PROGRAM SP_change
  VAR_OUTPUT
    wPrsHourSP_1 : WORD := 6;  (* Часы инициализации дневной уставки *)
    wPrsMinSP_1 : WORD;  (* Минуты инициализации дневной уставки *)
    wPrsHourSP_2 : WORD := 21;  (* Часы инициализации ночной уставки *)
    wPrsMinSP_2 : WORD;  (* Минуты инициализации ночной уставки *)
    wPrsHourSP_3 : WORD := 6;  (* Часы инициализации дневной зимней уставки *)
    wPrsMinSP_3 : WORD;  (* Минуты инициализации дневной зимней уставки *)
    wPrsHourSP_4 : WORD := 20;  (* Часы инициализации ночной зимней уставки *)
    wPrsMinSP_4 : WORD;  (* Минуты инициализации ночной зимней уставки *)
  END_VAR
  VAR_IN_OUT
    wPrsDayS : WORD;  (* День переключения на летний режим *)
    wPrsMonthS : WORD;  (* Месяц переключения на летний режим *)
    wPrsDayW : WORD;  (* День переключения на зимний режим *)
    wPrsMonthW : WORD;  (* Месяц переключения на зимний режим *)
  END_VAR
  VAR
    SP_in : REAL;  (* Входная уставка из контроллера *)
    SP_in2 : REAL;
    SP_old_man : REAL;
    write_sp : INT;
  END_VAR
  VAR_OUTPUT
    Summer : BOOL;
  END_VAR
  VAR_IN_OUT
    wCmdSP : WORD;  (* Слово на запись уставок *)
  END_VAR
  VAR_OUTPUT
    rPrsSP_1 : REAL;  (* Уставка давления №1 (летняя, дневная) *)
    rPrsSP_2 : REAL;  (* Уставка давления №2 (летняя, ночная) *)
    rPrsSP_3 : REAL;  (* Уставка давления №3 (зимняя, дневная) *)
    rPrsSP_4 : REAL;  (* Уставка давления №4 (зимняя, ночная) *)
    SP_target : REAL;
    SP : REAL;  (* Текущая уставка *)
  END_VAR
  VAR
    xPrsSP_N : BOOL;  (* Запись уставки по номеру *)
    xPrsSchedSP : BOOL;  (* Запись уставки по расписанию *)
    rem_auto_man : WORD := 3;  (* режим работы регулятора *)
    speed_limit : Speed_Lim;
    InputNum : Stat_to_num;
  END_VAR
  VAR_INPUT
    wNumSP : WORD;  (* Номер уставки *)
    rPrsDN : REAL;  (* Уставка давления день/ночь *)
    rPrsSched : REAL;  (* Уставка давления по расписанию *)
    rSP_manual : REAL;  (* Ручная уставка *)
    wPrsHourSP_N : WORD;  (* Часы инициализации уставки *)
    wPrsMinSP_N : WORD;  (* Минуты инициализации уставки *)
    xSCADA_Comm : BOOL;  (* Наличие связи со SCADA *)
    r_dSP : REAL;  (* скорость изменения уставки *)
  END_VAR

            wPrsMonthS:=LIMIT(1,wPrsMonthS,12);
wPrsMonthW:=LIMIT(1,wPrsMonthW,12);
wPrsDayS:=LIMIT(1, WORD_TO_UINT(wPrsDayS), QDay(y:=wYear , m:=WORD_TO_UINT(wPrsMonthS)));
wPrsDayW:=LIMIT(1, WORD_TO_UINT(wPrsDayW), QDay(y:=wYear , m:=WORD_TO_UINT(wPrsMonthW)));

IF wPrsMonthW > wPrsMonthS OR wPrsMonthW = wPrsMonthS AND wPrsDayW > wPrsDayS THEN
	IF wMonth>wPrsMonthW OR wMonth=wPrsMonthW AND wDay>=wPrsDayW OR wMonth<wPrsMonthS OR wMonth=wPrsMonthS AND wDay<wPrsDayS THEN
		Summer:=0;
		wCmdSP.10:=0;
	ELSIF wMonth>wPrsMonthS OR wMonth=wPrsMonthS AND wDay>=wPrsDayS THEN
		Summer:=1;
		wCmdSP.10:=1;
	END_IF
(*ELSE 
	END_IF*)
END_IF

///////////////////////////////Переключение уставок день/ночь/ Лето//////////////////////////
IF Summer THEN
IF wPrsHourSP_2>wPrsHourSP_1 OR wPrsHourSP_2=wPrsHourSP_1 AND wPrsMinSP_2>wPrsMinSP_1 THEN
	IF wHour>wPrsHourSP_2 OR wHour=wPrsHourSP_2 AND wMinute>=wPrsMinSP_2 OR wHour<wPrsHourSP_1 OR wHour=wPrsHourSP_1 AND wMinute<wPrsMinSP_1 THEN
		IF NOT write_sp.1 THEN
			write_sp:=0;
			SP_in:=rPrsSP_2;
			write_sp.1:=1;
		END_IF
	ELSIF wHour>wPrsHourSP_1 OR wHour=wPrsHourSP_1 AND wMinute>=wPrsMinSP_1 THEN
		IF NOT write_sp.0 THEN
			write_sp:=0;
			SP_in:=rPrsSP_1;
			write_sp.0:=1;
		END_IF
	END_IF
ELSE 
	IF wHour>wPrsHourSP_1 OR wHour=wPrsHourSP_1 AND wMinute>=wPrsMinSP_1 OR wHour<wPrsHourSP_2 OR wHour=wPrsHourSP_2 AND wMinute<wPrsMinSP_2 THEN
			IF NOT write_sp.2 THEN
			write_sp:=0;
			SP_in:=rPrsSP_1;
			write_sp.2:=1;
		END_IF
	ELSIF wHour>wPrsHourSP_2 OR wHour=wPrsHourSP_2 AND wMinute>=wPrsMinSP_2 THEN
		IF NOT write_sp.3 THEN
			write_sp:=0;
			SP_in:=rPrsSP_2;
			write_sp.3:=1;
		END_IF
	END_IF
END_IF
///////////////////////////////////////////////////////////////////////////////////////////////////
ELSE
///////////////////////////////Переключение уставок день/ночь/ Зима//////////////////////////
IF wPrsHourSP_4>wPrsHourSP_3 OR wPrsHourSP_4=wPrsHourSP_3 AND wPrsMinSP_4>wPrsMinSP_3 THEN
	IF wHour>wPrsHourSP_4 OR wHour=wPrsHourSP_4 AND wMinute>=wPrsMinSP_4 OR wHour<wPrsHourSP_3 OR wHour=wPrsHourSP_3 AND wMinute<wPrsMinSP_3 THEN
		IF NOT write_sp.5 THEN
			write_sp:=0;
			SP_in:=rPrsSP_4;
			write_sp.5:=1;
		END_IF
	ELSIF wHour>wPrsHourSP_3 OR wHour=wPrsHourSP_3 AND wMinute>=wPrsMinSP_3 THEN	
		IF NOT write_sp.4 THEN
			write_sp:=0;
			SP_in:=rPrsSP_3;
			write_sp.4:=1;
		END_IF
	END_IF
ELSE 
	IF wHour>wPrsHourSP_3 OR wHour=wPrsHourSP_3 AND wMinute>=wPrsMinSP_3 OR wHour<wPrsHourSP_4 OR wHour=wPrsHourSP_4 AND wMinute<wPrsMinSP_4 THEN
		IF NOT write_sp.6 THEN
			write_sp:=0;
			SP_in:=rPrsSP_3;
			write_sp.6:=1;
		END_IF
	ELSIF wHour>wPrsHourSP_4 OR wHour=wPrsHourSP_4 AND wMinute>=wPrsMinSP_4 THEN
		IF NOT write_sp.7 THEN
			write_sp:=0;
			SP_in:=rPrsSP_4;
			write_sp.7:=1;
		END_IF
	END_IF
END_IF
///////////////////////////////////////////////////////////////////////////////////////////////////
END_IF;

InputNum(in1:=wCmdSP.3,in2:=wCmdSP.4,in3:=wCmdSP.5);
rem_auto_man:=InputNum.out;

///////////////////////////////Ввод уставок из SCADA///////////////////////////
xPrsSP_N:=wCmdSP.0;
	IF xPrsSP_N THEN
		CASE wNumSP OF
			1: rPrsSP_1:=rPrsDN;
			wPrsHourSP_1:=wPrsHourSP_N;
			wPrsMinSP_1:=wPrsMinSP_N;
			2: rPrsSP_2:=rPrsDN;
			wPrsHourSP_2:=wPrsHourSP_N;
			wPrsMinSP_2:=wPrsMinSP_N;						
			3: rPrsSP_3:=rPrsDN;
			wPrsHourSP_3:=wPrsHourSP_N;
			wPrsMinSP_3:=wPrsMinSP_N;			
			4: rPrsSP_4:=rPrsDN;
			wPrsHourSP_4:=wPrsHourSP_N;
			wPrsMinSP_4:=wPrsMinSP_N;
		END_CASE
		xPrsSP_N:=0;
		wCmdSP.0:=0;
	END_IF
xPrsSchedSP:=wCmdSP.1;
	IF xPrsSchedSP THEN
		SP_in2:=rPrsSched;
		xPrsSchedSP:=0;
		wCmdSP.1:=0;
	END_IF
CASE rem_auto_man OF 
	1: SP_target:=rSP_manual;
	2: SP_target:=SP_in;
	3: IF xSCADA_Comm THEN
		SP_target:=SP_in2;	
		ELSE
		SP_target:=SP_in;
		END_IF;
END_CASE;
IF rSP_manual <> SP_old_man THEN
	CASE rem_auto_man OF 
		2: SP_in:=rSP_manual;
		3: SP_in2:=rSP_manual;
			SP_in:=rSP_manual;
	END_CASE;
	SP_old_man:=rSP_manual;
END_IF;
speed_limit(SP_target:= SP_target, dSP:= r_dSP, PLC_Cycle:= PLC_Cycle, Translate:= 1);
SP:=speed_limit.SP;

          
END_PROGRAM

FUNCTION LeapYear : BOOL
  VAR_INPUT
    y : WORD;
  END_VAR

            LeapYear:= y MOD 400 = 0 OR y MOD 4 = 0 OR y MOD 100 <>0;

          
END_FUNCTION

FUNCTION QDay : UINT
  VAR_INPUT
    y : UINT;
    m : UINT;
  END_VAR
  VAR CONSTANT
    dpm : ARRAY[1..12] OF UINT := [31, 28, 31, 30, 31, 30, 31, 31, 30, 31, 30, 31];
  END_VAR

            m:= LIMIT(1,m,12);
QDay:= dpm[m] + BOOL_TO_UINT(m=2 AND LeapYear(y));

          
END_FUNCTION

FUNCTION swap_byte : DWORD
  VAR_INPUT
    IN : DWORD;
    Mode : INT;
  END_VAR

            CASE Mode OF
1:swap_byte:=(ROR(IN,16)); 													// MEM.ReverseWORDsInDWORD
2:swap_byte := (ROR(IN,8) AND 16#00FF00FF) OR (ROL(IN,8) AND 16#FF00FF00); 	// AABB CCDD => BBAA DDCC
3:swap_byte := (ROR(IN,8) AND 16#FF00FF00) OR (ROL(IN,8) AND 16#00FF00FF); 	// AABB CCDD => DDCC BBAA   MEM.ReverseBYTEsInDWORD
END_CASE

          
END_FUNCTION

FUNCTION_BLOCK Power_c
  VAR_IN_OUT
    PM_FB : FB_PowerMeter;
  END_VAR
  VAR
    FB_ERR : Comm_error;
    xEnable : BOOL;
    xReset : BOOL;
    dataset : EET.ST_GenericDeviceDatasetLong;
    rCur_A1 : REAL;
    pntr : POINTER TO WORD;
    highwrd : WORD;
    lowwrd1 : WORD;
    highwrd1 : WORD;
    lowwrd2 : WORD;
    highwrd2 : WORD;
    highwrd3 : WORD;
    lowwrd3 : WORD;
    lowwrd4 : WORD;
    highwrd4 : WORD;
  END_VAR
  VAR_OUTPUT
    x_alarm_comm : BOOL;
    rCurA : REAL;
    rCurB : REAL;
    rCurC : REAL;
    rCurAvg : REAL;
    rVol12 : REAL;
    rVol23 : REAL;
    rVol31 : REAL;
    rVolAvg : REAL;
    rTotPwrA : REAL;  (* Мощность активная *)
    rTotPwrR : REAL;  (* Мощность реактивная *)
    rTotPwrAp : REAL;  (* apparent power полная мощность *)
    rPwrFact : REAL;
    rCurFrq : REAL;
    rEnergyA : REAL;
    rEnergyR : REAL;
    rEnergyA_L : DWORD;
    rEnergyA_H : DWORD;
    rEnergyR_L : DWORD;
    rEnergyR_H : DWORD;
  END_VAR
  VAR
    x_set_measure : BOOL;
    w_Token : WORD;
  END_VAR
  VAR_INPUT
    com_err : INT;
    modbus_slave_ch6 : POINTER TO ARRAY[0..7] OF WORD;
  END_VAR

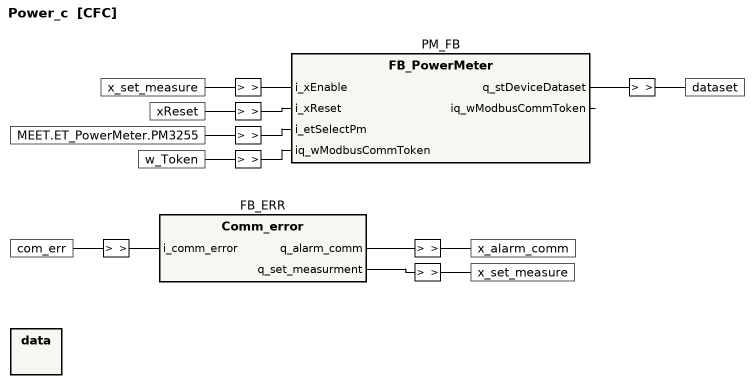
(* CFC diagram, written out as Structured Text *)
PM_FB(i_xEnable := x_set_measure, i_xReset := xReset, i_etSelectPm := MEET.ET_PowerMeter.PM3255, iq_wModbusCommToken := w_Token);
dataset := PM_FB.q_stDeviceDataset;
data();
FB_ERR(i_comm_error := com_err);
x_alarm_comm := FB_ERR.q_alarm_comm;
x_set_measure := FB_ERR.q_set_measurment;

ACTION data:
                rCurA:=dataset.stCurrent.rLine1;
rCurB:=dataset.stCurrent.rLine2;
rCurC:=dataset.stCurrent.rLine3;
rCurAvg:=dataset.stCurrent.rAverage;
rVol12:=dataset.stVoltage.rLine12;
rVol23:=dataset.stVoltage.rLine23;
rVol31:=dataset.stVoltage.rLine31;
rVolAvg:=dataset.stVoltage.rLineLavg;
// Мощность активная
rTotPwrA:=dataset.stPower.rReTotal/1000;
// Мощность реактивная
rTotPwrR:=dataset.stPower.rRvTotal/1000;
// apparent power  полная мощность
rTotPwrAp:=dataset.stPower.rApTotal/1000;
rPwrFact:=dataset.stPowerFactor.rTotal;
rCurFrq:=dataset.stFrequency.rFrequency;
rEnergyA:=dataset.stEnergy.rReal;
rEnergyR:=dataset.stEnergy.rRctv;


lowwrd1:=modbus_slave_ch6^[0];
highwrd1:=modbus_slave_ch6^[1];
rEnergyA_H:=MEM.PackWordsToDword(highwrd1,lowwrd1);
lowwrd2:=modbus_slave_ch6^[2];
highwrd2:=modbus_slave_ch6^[3];
rEnergyA_L:=MEM.PackWordsToDword(highwrd2,lowwrd2);
lowwrd3:=modbus_slave_ch6^[4];
highwrd3:=modbus_slave_ch6^[5];
rEnergyR_H:=MEM.PackWordsToDword(highwrd3,lowwrd3);
lowwrd4:=modbus_slave_ch6^[6];
highwrd4:=modbus_slave_ch6^[7];
rEnergyR_L:=MEM.PackWordsToDword(highwrd4,lowwrd4);


              
END_ACTION
END_FUNCTION_BLOCK

FUNCTION_BLOCK dPos_to_timesetup
  VAR_INPUT
    open : BOOL;
    close : BOOL;
  END_VAR
  VAR_OUTPUT
    pos : REAL;
  END_VAR
  VAR
    dpos : REAL;
  END_VAR
  VAR_INPUT
    time_move : TIME;
  END_VAR

            	//dpos:=TIME_TO_INT
	dpos:=(100/(TIME_TO_REAL(time_move)/1000))*PLC_Cycle;
	IF open AND pos < 100 THEN
		IF ABS(100-pos) >= dpos THEN
			pos:=pos+dpos;
		ELSE
			pos:=100;
		END_IF;
	END_IF;
	IF close AND pos > 0 THEN
		IF ABS(pos) >= dpos THEN
			pos:=pos-dpos;
		ELSE
			pos:=0;
		END_IF;
	END_IF;
          
END_FUNCTION_BLOCK

(* Converting DWORD to REAL (FLOAT32) *)
FUNCTION Dw_to_real : REAL
  VAR_INPUT
    IN : DWORD;
  END_VAR
  VAR
    pr : POINTER TO REAL;
  END_VAR

            pr:= ADR(IN);
Dw_to_real:= pr^;
          
END_FUNCTION

FUNCTION_BLOCK Analog_Input
  VAR_INPUT
    i_sensor_value : INT;
    i_status_analog : BYTE;
    k : REAL;
    b : REAL;
    i_ADC_Range : INT;
  END_VAR
  VAR_OUTPUT
    q_Out : REAL;
    q_status_analog : BYTE;
    xAlarm_bit : BOOL;
  END_VAR

            q_Out:=k*INT_TO_REAL(i_sensor_value)/INT_TO_REAL(i_ADC_Range)+b;
q_status_analog:=i_status_analog;

IF q_status_analog=0 THEN
xAlarm_bit:=0;
ELSE
	IF q_status_analog>0 THEN
		xAlarm_bit:=1;	
	END_IF;
END_IF;
          
END_FUNCTION_BLOCK

PROGRAM SetPointSect
  VAR
    ConectCheck : TOF;
    wWinDate : WORD;
    wSummDate : WORD;
    wCurrDate : WORD;
    wSummDayTime : WORD;
    wSummNightTime : WORD;
    wWinDayTime : WORD;
    wWinNightTime : WORD;
    wCurrTime : WORD;
    xSummer : BOOL;
    xWinter : BOOL;
    i : INT;
    xSchedPLS : R_TRIG;
    xSchedSP1_PLS : R_TRIG;
    xSchedSP2_PLS : R_TRIG;
    xSchedSP3_PLS : R_TRIG;
    xSchedSP4_PLS : R_TRIG;
    xRemotePLS : R_TRIG;
    xRemoteSetPLS : R_TRIG;
    xRemoteNoConnPLS : R_TRIG;
  END_VAR

            // Date input restriction
SetPoint.sSPDate.wSummMonth:= LIMIT(1, SetPoint.sSPDate.wSummMonth, 12);
SetPoint.sSPDate.wWinMonth:= LIMIT(1, SetPoint.sSPDate.wWinMonth, 12);
SetPoint.sSPDate.wSummDay:= LIMIT(1, SetPoint.sSPDate.wSummDay, 31);
SetPoint.sSPDate.wWinDay:= LIMIT(1, SetPoint.sSPDate.wWinDay, 31);

// Convert the date of type “mm:dd” to a number
wSummDate:= (SetPoint.sSPDate.wSummMonth * 100) + SetPoint.sSPDate.wSummDay;
wWinDate:= (SetPoint.sSPDate.wWinMonth * 100) + SetPoint.sSPDate.wWinDay;
wCurrDate:= (PLC_RTC.wMonth * 100) + PLC_RTC.wDay;

// Defining the summer period
xSummer:= ((wCurrDate >= wSummDate) AND (wCurrDate < wWinDate)) OR ((wSummDate > wWinDate) AND ((wCurrDate >= wSummDate) OR (wCurrDate < wWinDate)));
// Defining the winter period
xWinter:= (wCurrDate >= wWinDate) AND (wCurrDate < wSummDate) OR ((wWinDate > wSummDate) AND ((wCurrDate >= wWinDate) OR (wCurrDate < wSummDate)));




// Recording time and setpoints in the schedule
IF SetPoint.CW.xSPLocSet THEN
	SetPoint.arrSPLocCurr[SetPoint.wSPLocSetNum].wHour:= SetPoint.sSPLocSet.wHour;
	SetPoint.arrSPLocCurr[SetPoint.wSPLocSetNum].wMinute:= SetPoint.sSPLocSet.wMinute;
	SetPoint.arrSPLocCurr[SetPoint.wSPLocSetNum].rSP:= SetPoint.sSPLocSet.rSP;
	SetPoint.CW.xSPLocSet:= FALSE;
END_IF

// Time entry restriction 
SetPoint.sSPLocSet.wHour:= LIMIT(0, SetPoint.sSPLocSet.wHour, 24);
SetPoint.sSPLocSet.wMinute:= LIMIT(0, SetPoint.sSPLocSet.wMinute, 59);
FOR i:= 1 TO 4 DO
	SetPoint.arrSPLocCurr[i].wHour:= LIMIT(0, SetPoint.arrSPLocCurr[i].wHour, 24);
	SetPoint.arrSPLocCurr[i].wMinute:= LIMIT(0, SetPoint.arrSPLocCurr[i].wMinute, 59);
END_FOR

// Convert time type “hh:mm” to a number
wSummDayTime:= (SetPoint.arrSPLocCurr[1].wHour * 100) + SetPoint.arrSPLocCurr[1].wMinute; 
wSummNightTime:= (SetPoint.arrSPLocCurr[2].wHour * 100) + SetPoint.arrSPLocCurr[2].wMinute; 
wWinDayTime:= (SetPoint.arrSPLocCurr[3].wHour * 100) + SetPoint.arrSPLocCurr[3].wMinute; 
wWinNightTime:= (SetPoint.arrSPLocCurr[4].wHour * 100) + SetPoint.arrSPLocCurr[4].wMinute;
wCurrTime:= (PLC_RTC.wHour * 100) + PLC_RTC.wMinute; 

// Determine the day and night time of the summer period and set the corresponding setpoint number
IF xSummer THEN
	IF ((wCurrTime >= wSummDayTime) AND (wCurrTime < wSummNightTime)) OR ((wSummDayTime > wSummNightTime) AND ((wCurrTime >= wSummDayTime) OR (wCurrTime < wSummNightTime))) THEN
		SetPoint.wSPLocCurrNum:= 1;
	ELSIF ((wCurrTime >= wSummNightTime) AND (wCurrTime < wSummDayTime)) OR ((wSummNightTime > wSummDayTime) AND ((wCurrTime >= wSummNightTime) OR (wCurrTime < wSummDayTime))) THEN
		SetPoint.wSPLocCurrNum:= 2;
	END_IF
END_IF

// Determine the day and night time of the winter period and set the corresponding setpoint number
IF xWinter THEN
	IF ((wCurrTime >= wWinDayTime) AND (wCurrTime < wWinNightTime)) OR ((wWinDayTime > wWinNightTime) AND ((wCurrTime >= wWinDayTime) OR (wCurrTime < wWinNightTime))) THEN
		SetPoint.wSPLocCurrNum:= 3;
	ELSIF ((wCurrTime >= wWinNightTime) AND (wCurrTime < wWinDayTime)) OR ((wWinNightTime > wWinDayTime) AND ((wCurrTime >= wWinNightTime) OR (wCurrTime < wWinDayTime))) THEN
		SetPoint.wSPLocCurrNum:= 4;
	END_IF
END_IF




IF SetPoint.CW.xManMode THEN															// Selecting the manual setpoint mode											
	SetPoint.SW.xManual:= TRUE;
	SetPoint.SW.xSched:= FALSE;
	SetPoint.SW.xRemote:= FALSE;
	SetPoint.CW.xManMode:= FALSE;
ELSIF SetPoint.CW.xAutoLocMode THEN														// Selecting the automatic setpoint mode											
	SetPoint.SW.xManual:= FALSE;
	SetPoint.SW.xSched:= TRUE;
	SetPoint.SW.xRemote:= FALSE;
	SetPoint.CW.xAutoLocMode:= FALSE;
ELSIF SetPoint.CW.xAutoRemMode THEN														// Selecting the automatic remote setpoint mode											
	SetPoint.SW.xManual:= FALSE;
	SetPoint.SW.xSched:= FALSE;
	SetPoint.SW.xRemote:= TRUE;
	SetPoint.CW.xAutoRemMode:= FALSE;
ELSIF NOT SetPoint.SW.xManual AND NOT SetPoint.SW.xSched AND NOT SetPoint.SW.xRemote THEN
	SetPoint.SW.xSched:= TRUE;
END_IF 

// SCADA communication check
ConectCheck(IN:= SetPoint.CW.xConnect OR SetPoint.wConnect.2, PT:= T#3M); 	

xSchedPLS(CLK:= SetPoint.SW.xSched);																				// Pulse to switch to schedule mode
xSchedSP1_PLS(CLK:= SetPoint.SW.xSched AND (SetPoint.wSPLocCurrNum = 1));											// Pulse of the 1st setpoint on schedule
xSchedSP2_PLS(CLK:= SetPoint.SW.xSched AND (SetPoint.wSPLocCurrNum = 2));											// Pulse of the 2nd setpoint on schedule
xSchedSP3_PLS(CLK:= SetPoint.SW.xSched AND (SetPoint.wSPLocCurrNum = 3));											// Pulse of the 3rd setpoint on schedule
xSchedSP4_PLS(CLK:= SetPoint.SW.xSched AND (SetPoint.wSPLocCurrNum = 4));											// Pulse of the 4th setpoint on schedule

xRemotePLS(CLK:= SetPoint.SW.xRemote);																				// Remote mode transition pulse
xRemoteSetPLS(CLK:= SetPoint.SW.xRemote AND ConectCheck.Q AND (SetPoint.CW.xSPRemSet OR SetPoint.wSPRemSet.2));		// Remote setpoint change pulse
xRemoteNoConnPLS(CLK:= SetPoint.SW.xRemote AND NOT ConectCheck.Q);													// Pulse of SCADA communication loss


IF xSchedPLS.Q OR xSchedSP1_PLS.Q OR xSchedSP2_PLS.Q OR xSchedSP3_PLS.Q OR xSchedSP4_PLS.Q OR xRemoteNoConnPLS.Q THEN
	Cycle.rSP:= SetPoint.arrSPLocCurr[SetPoint.wSPLocCurrNum].rSP;													// Setting the setpoint by schedule
ELSIF xRemotePLS.Q OR xRemoteSetPLS.Q THEN
	Cycle.rSP:= SetPoint.rSPRem;																					// Setpoint setting remotely
END_IF

IF SetPoint.wSPRemSet.2 THEN
	SetPoint.wSPRemSet.2:= FALSE;
END_IF

IF SetPoint.CW.xSPRemSet THEN
	SetPoint.CW.xSPRemSet:= FALSE;
END_IF




          
END_PROGRAM
